// TIA Portal V20 export
// export: Created 2025-12-01T14:56:56.3805468Z, ExportSetting None, DisplayName Totally Integrated Automation Portal, DisplayVersion V20 Update 3, DisplayName TIA Portal Openness, DisplayVersion V20 Update 3, DisplayName TIA Portal Version Control Interface, DisplayVersion V20 Update 3, DisplayName STEP 7 Professional, DisplayVersion V20 Update 3, DisplayName STEP 7 Safety, DisplayVersion V20 Update 2, DisplayName WinCC Basic/Comfort/Advanced, DisplayVersion V20 Update 3, DisplayName WinCC Professional, DisplayVersion V20 Update 3, DisplayName WinCC Unified, DisplayVersion V20 Update 3
FUNCTION_BLOCK "FB490_ControlEtiquetadora_ZETES"   // FB490, LAD
{ S7_Optimized_Access := 'FALSE' }
// stored: AutoNumber false, SetENOAutomatically false
   VAR_INPUT
      NumMaquina : UInt;   // Numero de Maquina
      NumMesa : UInt;
      In_PowerOn : Bool;
      In_Online : Bool;
      In_Consumible : Bool;
      In_Bypass : Bool;
      In_BrazoRecogido : Bool;
      In_DataReady : Bool;
      In_FinCiclo : Bool;
   END_VAR
   VAR_OUTPUT
      Out_InicioCiclo : Bool;
      Parar_Tx { ExternalAccessible := 'False'; ExternalVisible := 'False'; ExternalWritable := 'False'} : Bool;
   END_VAR
   VAR
      Mx_ET00 : Bool;
      Mx_ET01 : Bool;
      Mx_ET02 : Bool;
      Mx_ET03 : Bool;
      Mx_ET04 : Bool;
      Mx_ET05 : Bool;
      Mx_ET06 : Bool;
      Mx_ET07 : Bool;
      EmpezandoProceso : Bool;
      FinalProceso : Bool;
      ErrorProceso : Bool;
      Interlock_manual { S7_SetPoint := 'True'} : "UDT_Interlock_manual_Etiquetadora";
   END_VAR
   VAR_TEMP
      VarEventos : Struct
         NumeroUT : UInt;
         ProcesoActual : UInt;
         P_EmiEventos : DWord;
         DBEventos : Word;
         NumDBEventos : UInt;
         MaxBytes : UInt;
         NumBytes : UInt;
         OffsetInicial : UInt;
         OffsetFinal : UInt;
         Conversion : DWord;
         Convertir : UInt;
         Valor : UDInt;
      END_STRUCT;
      Informe_disp_maquina : "UDT_Informe_DispositivoMaquina";
      Interlock : "UDT_Interlock_Etiquetadora_ZETES";
      retval : Int;
      cero : USInt;
      Etiq_Online : Bool;
      Etiq_Error : Bool;
      OrdenDeEtiquetar : Bool;
      Reset : Bool;
   END_VAR
   VAR_TEMP   // added for the SCL form of the ladder/FBD networks
      _w1 : Bool;
   END_VAR
BEGIN

REGION Network 1: INICIALIZAR
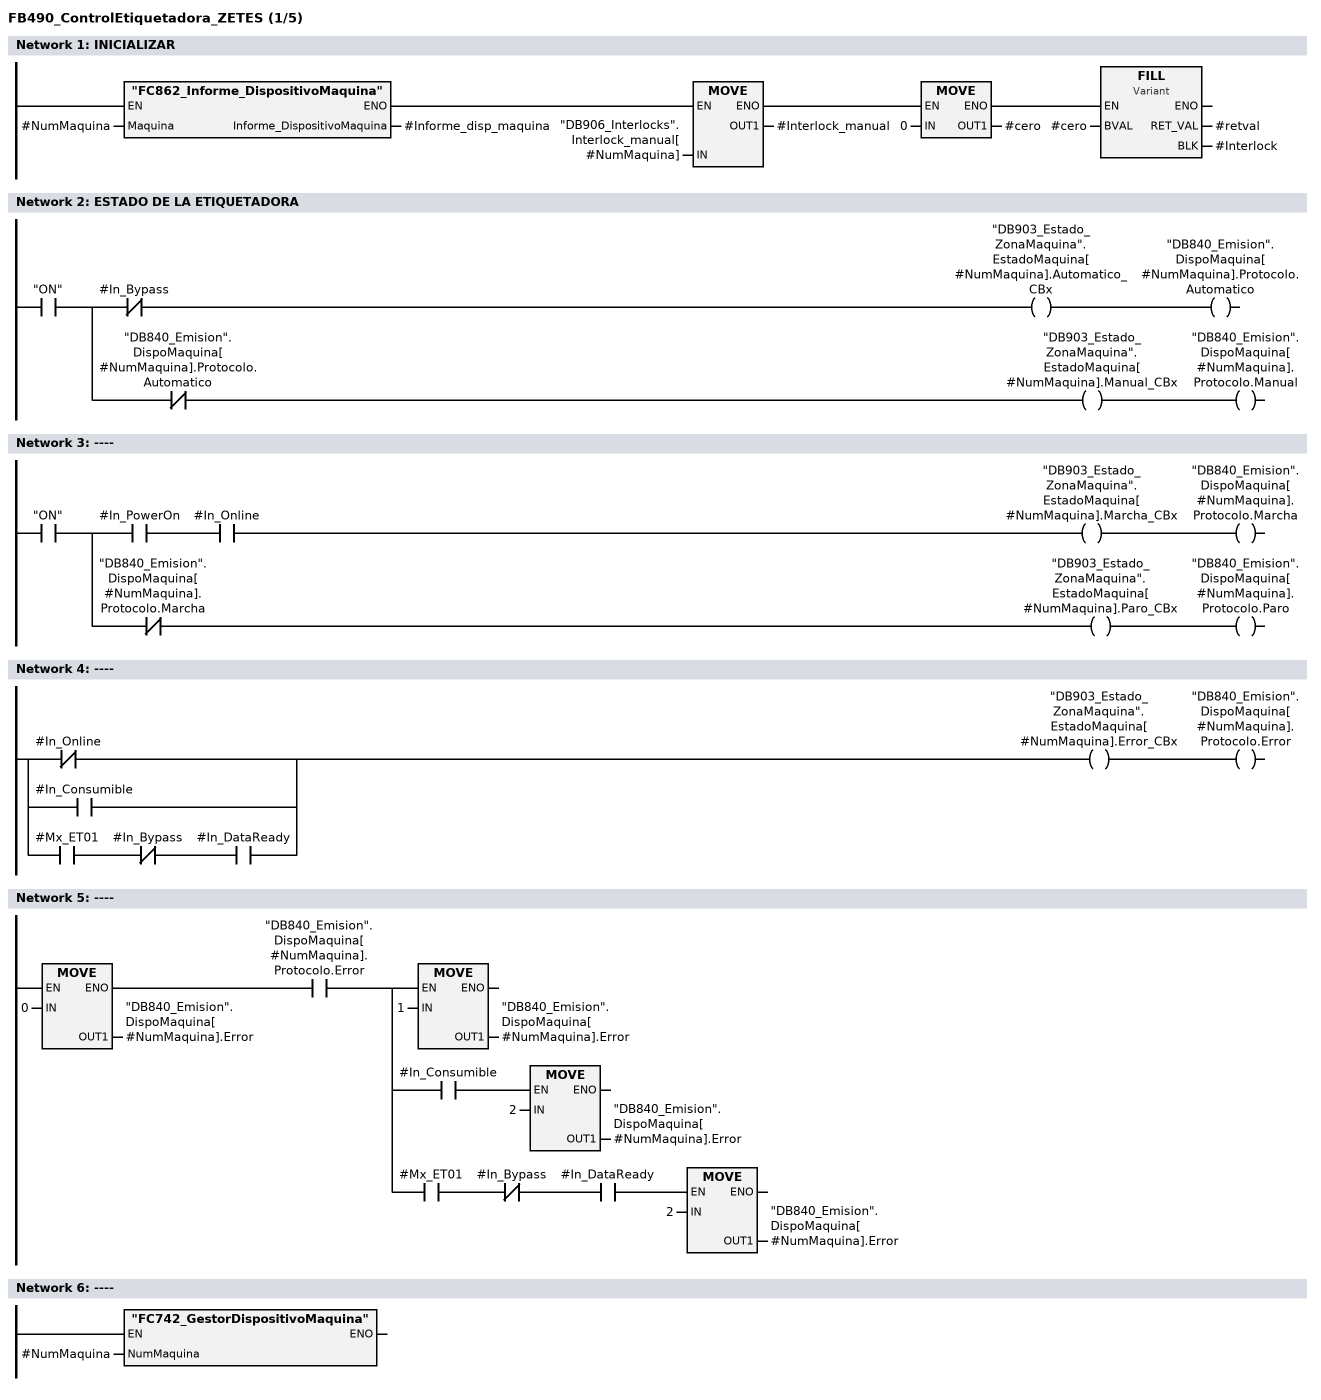
   RUNG wire#powerrail
      "FC862_Informe_DispositivoMaquina"(Maquina := #NumMaquina, Informe_DispositivoMaquina => #Informe_disp_maquina)
      Move(in := "DB906_Interlocks".Interlock_manual[#NumMaquina], out1 => #Interlock_manual)
      Move(in := 0, out1 => #cero)
      { S7_Templates := "ptr_type := Variant" } FILL(BVAL := #cero, RET_VAL => #retval, BLK => #Interlock)
   END_RUNG
   // the same network as SCL:
   "FC862_Informe_DispositivoMaquina"(Maquina := #NumMaquina,
                           Informe_DispositivoMaquina => #Informe_disp_maquina,
                           ENO => #_w1);
   IF #_w1 THEN
       #Interlock_manual := "DB906_Interlocks".Interlock_manual[#NumMaquina];
       #cero := 0;
       #retval := FILL(BVAL := #cero, BLK => #Interlock);
   END_IF;
END_REGION

REGION Network 2: ESTADO DE LA ETIQUETADORA
   RUNG wire#powerrail
      Contact( "ON" )
      wire#w1
      I_Contact( #In_Bypass )
      Coil( "DB903_Estado_ZonaMaquina".EstadoMaquina[#NumMaquina].Automatico_CBx )
      Coil( "DB840_Emision".DispoMaquina[#NumMaquina].Protocolo.Automatico )
   END_RUNG
   RUNG wire#w1
      I_Contact( "DB840_Emision".DispoMaquina[#NumMaquina].Protocolo.Automatico )
      Coil( "DB903_Estado_ZonaMaquina".EstadoMaquina[#NumMaquina].Manual_CBx )
      Coil( "DB840_Emision".DispoMaquina[#NumMaquina].Protocolo.Manual )
   END_RUNG
   // the same network as SCL:
   "DB903_Estado_ZonaMaquina".EstadoMaquina[#NumMaquina].Automatico_CBx := "ON" AND NOT #In_Bypass;
   "DB840_Emision".DispoMaquina[#NumMaquina].Protocolo.Automatico := "ON" AND NOT #In_Bypass;
   #_w1 := "ON" AND NOT "DB840_Emision".DispoMaquina[#NumMaquina].Protocolo.Automatico;
   "DB903_Estado_ZonaMaquina".EstadoMaquina[#NumMaquina].Manual_CBx := #_w1;
   "DB840_Emision".DispoMaquina[#NumMaquina].Protocolo.Manual := #_w1;
END_REGION

REGION Network 3: ----
   RUNG wire#powerrail
      Contact( "ON" )
      wire#w1
      Contact( #In_PowerOn )
      Contact( #In_Online )
      Coil( "DB903_Estado_ZonaMaquina".EstadoMaquina[#NumMaquina].Marcha_CBx )
      Coil( "DB840_Emision".DispoMaquina[#NumMaquina].Protocolo.Marcha )
   END_RUNG
   RUNG wire#w1
      I_Contact( "DB840_Emision".DispoMaquina[#NumMaquina].Protocolo.Marcha )
      Coil( "DB903_Estado_ZonaMaquina".EstadoMaquina[#NumMaquina].Paro_CBx )
      Coil( "DB840_Emision".DispoMaquina[#NumMaquina].Protocolo.Paro )
   END_RUNG
   // the same network as SCL:
   "DB903_Estado_ZonaMaquina".EstadoMaquina[#NumMaquina].Marcha_CBx := "ON" AND #In_PowerOn AND #In_Online;
   "DB840_Emision".DispoMaquina[#NumMaquina].Protocolo.Marcha := "ON" AND #In_PowerOn AND #In_Online;
   #_w1 := "ON" AND NOT "DB840_Emision".DispoMaquina[#NumMaquina].Protocolo.Marcha;
   "DB903_Estado_ZonaMaquina".EstadoMaquina[#NumMaquina].Paro_CBx := #_w1;
   "DB840_Emision".DispoMaquina[#NumMaquina].Protocolo.Paro := #_w1;
END_REGION

REGION Network 4: ----
   RUNG wire#powerrail
      I_Contact( #In_Online )
      wire#w1
      Coil( "DB903_Estado_ZonaMaquina".EstadoMaquina[#NumMaquina].Error_CBx )
      Coil( "DB840_Emision".DispoMaquina[#NumMaquina].Protocolo.Error )
   END_RUNG
   RUNG wire#powerrail
      Contact( #In_Consumible )
   END_RUNG wire#w1
   RUNG wire#powerrail
      Contact( #Mx_ET01 )
      I_Contact( #In_Bypass )
      Contact( #In_DataReady )
   END_RUNG wire#w1
   // the same network as SCL:
   "DB903_Estado_ZonaMaquina".EstadoMaquina[#NumMaquina].Error_CBx := NOT #In_Online OR #In_Consumible OR (#Mx_ET01 AND NOT #In_Bypass AND #In_DataReady);
   "DB840_Emision".DispoMaquina[#NumMaquina].Protocolo.Error := NOT #In_Online OR #In_Consumible OR (#Mx_ET01 AND NOT #In_Bypass AND #In_DataReady);
END_REGION

REGION Network 5: ----
   RUNG wire#powerrail
      Move(in := 0, out1 => "DB840_Emision".DispoMaquina[#NumMaquina].Error)
      Contact( "DB840_Emision".DispoMaquina[#NumMaquina].Protocolo.Error )
      wire#w1
      Move(in := 1, out1 => "DB840_Emision".DispoMaquina[#NumMaquina].Error)
   END_RUNG
   RUNG wire#w1
      Contact( #In_Consumible )
      Move(in := 2, out1 => "DB840_Emision".DispoMaquina[#NumMaquina].Error)
   END_RUNG
   RUNG wire#w1
      Contact( #Mx_ET01 )
      I_Contact( #In_Bypass )
      Contact( #In_DataReady )
      Move(in := 2, out1 => "DB840_Emision".DispoMaquina[#NumMaquina].Error)
   END_RUNG
   // the same network as SCL:
   "DB840_Emision".DispoMaquina[#NumMaquina].Error := 0;
   #_w1 := "DB840_Emision".DispoMaquina[#NumMaquina].Protocolo.Error;
   IF #_w1 THEN "DB840_Emision".DispoMaquina[#NumMaquina].Error := 1; END_IF;
   IF #_w1 AND #In_Consumible THEN "DB840_Emision".DispoMaquina[#NumMaquina].Error := 2; END_IF;
   IF #_w1 AND #Mx_ET01 AND NOT #In_Bypass AND #In_DataReady THEN
       "DB840_Emision".DispoMaquina[#NumMaquina].Error := 2;
   END_IF;
END_REGION

REGION Network 6: ----
   RUNG wire#powerrail
      "FC742_GestorDispositivoMaquina"(NumMaquina := #NumMaquina)
   END_RUNG
   // the same network as SCL:
   "FC742_GestorDispositivoMaquina"(NumMaquina := #NumMaquina);
END_REGION

REGION Network 7: VARIABLES INTERNAS - Etiquetadora en ONLINE / ERROR
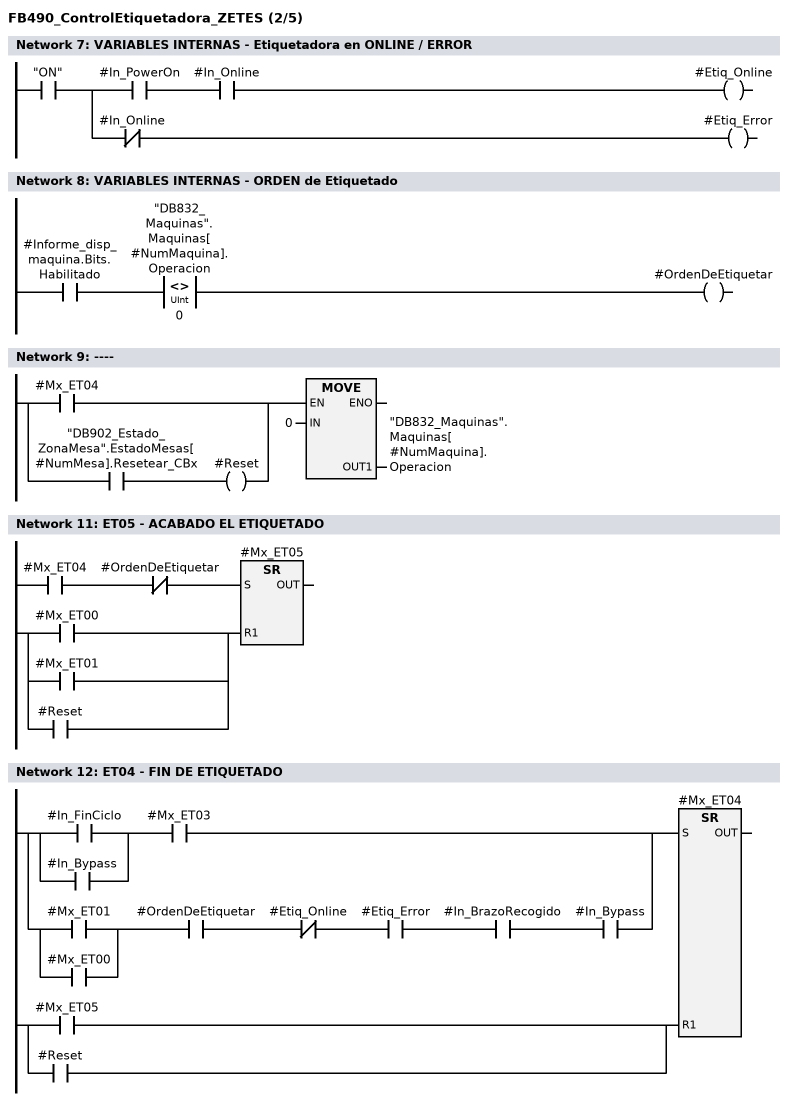
   RUNG wire#powerrail
      Contact( "ON" )
      wire#w1
      Contact( #In_PowerOn )
      Contact( #In_Online )
      Coil( #Etiq_Online )
   END_RUNG
   RUNG wire#w1
      I_Contact( #In_Online )
      Coil( #Etiq_Error )
   END_RUNG
   // the same network as SCL:
   #Etiq_Online := "ON" AND #In_PowerOn AND #In_Online;
   #Etiq_Error := "ON" AND NOT #In_Online;
END_REGION

REGION Network 8: VARIABLES INTERNAS - ORDEN de Etiquetado
   RUNG wire#powerrail
      Contact( #Informe_disp_maquina.Bits.Habilitado )
      { S7_Templates := "SrcType := UInt" } NE_Contact(in1 := "DB832_Maquinas".Maquinas[#NumMaquina].Operacion, in2 := 0)
      Coil( #OrdenDeEtiquetar )
   END_RUNG
   // the same network as SCL:
   #OrdenDeEtiquetar := #Informe_disp_maquina.Bits.Habilitado AND ("DB832_Maquinas".Maquinas[#NumMaquina].Operacion <> 0);
END_REGION

REGION Network 9: ----
   RUNG wire#powerrail
      Contact( #Mx_ET04 )
      wire#w1
      Move(in := 0, out1 => "DB832_Maquinas".Maquinas[#NumMaquina].Operacion)
   END_RUNG
   RUNG wire#powerrail
      Contact( "DB902_Estado_ZonaMesa".EstadoMesas[#NumMesa].Resetear_CBx )
      Coil( #Reset )
   END_RUNG wire#w1
   // the same network as SCL:
   #Reset := "DB902_Estado_ZonaMesa".EstadoMesas[#NumMesa].Resetear_CBx;
   IF #Mx_ET04 OR "DB902_Estado_ZonaMesa".EstadoMesas[#NumMesa].Resetear_CBx THEN
       "DB832_Maquinas".Maquinas[#NumMaquina].Operacion := 0;
   END_IF;
END_REGION

REGION Network 10: >>>>>>>>>>>>>>>>>>>>>>>>>>>>>>>>>>>>>>>>>>>>>>>>>>>>>>>>>>>>>>>>>>>>>>>>>>>>>>>>>>>>>>>>>>>>>>>
END_REGION

REGION Network 11: ET05 - ACABADO EL ETIQUETADO
   RUNG wire#powerrail
      Contact( #Mx_ET04 )
      I_Contact( #OrdenDeEtiquetar )
      S_SR(operand := #Mx_ET05, r1 := wire#w1)
   END_RUNG
   RUNG wire#powerrail
      Contact( #Mx_ET00 )
   END_RUNG wire#w1
   RUNG wire#powerrail
      Contact( #Mx_ET01 )
   END_RUNG wire#w1
   RUNG wire#powerrail
      Contact( #Reset )
   END_RUNG wire#w1
   // the same network as SCL:
   IF #Mx_ET04 AND NOT #OrdenDeEtiquetar THEN
       #Mx_ET05 := TRUE;   // SR flip-flop
   END_IF;
   IF #Mx_ET00 OR #Mx_ET01 OR #Reset THEN #Mx_ET05 := FALSE; END_IF;
END_REGION

REGION Network 12: ET04 - FIN DE ETIQUETADO
   RUNG wire#powerrail
      Contact( #In_FinCiclo )
      wire#w1
      Contact( #Mx_ET03 )
      wire#w2
      S_SR(operand := #Mx_ET04, r1 := wire#w4)
   END_RUNG
   RUNG wire#powerrail
      Contact( #In_Bypass )
   END_RUNG wire#w1
   RUNG wire#powerrail
      Contact( #Mx_ET01 )
      wire#w3
      Contact( #OrdenDeEtiquetar )
      I_Contact( #Etiq_Online )
      Contact( #Etiq_Error )
      Contact( #In_BrazoRecogido )
      Contact( #In_Bypass )
   END_RUNG wire#w2
   RUNG wire#powerrail
      Contact( #Mx_ET00 )
   END_RUNG wire#w3
   RUNG wire#powerrail
      Contact( #Mx_ET05 )
   END_RUNG wire#w4
   RUNG wire#powerrail
      Contact( #Reset )
   END_RUNG wire#w4
   // the same network as SCL:
   IF ((#In_FinCiclo OR #In_Bypass) AND #Mx_ET03) OR ((#Mx_ET01 OR #Mx_ET00) AND #OrdenDeEtiquetar AND NOT #Etiq_Online AND #Etiq_Error AND #In_BrazoRecogido AND #In_Bypass) THEN
       #Mx_ET04 := TRUE;   // SR flip-flop
   END_IF;
   IF #Mx_ET05 OR #Reset THEN #Mx_ET04 := FALSE; END_IF;
END_REGION

REGION Network 13: ET03 - ETIQUETANDO
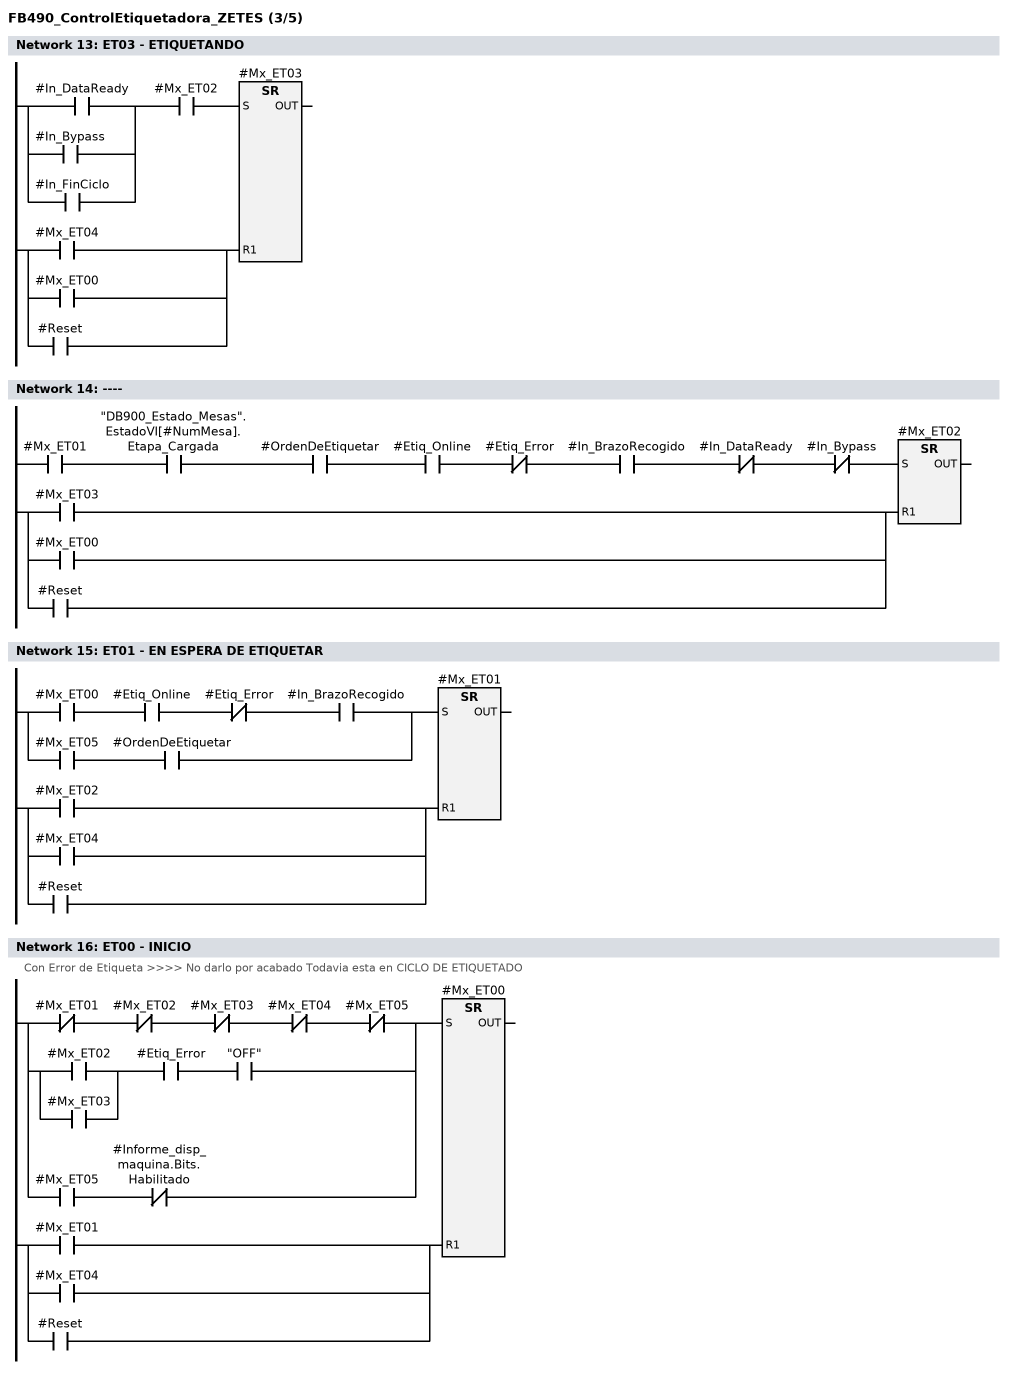
   RUNG wire#powerrail
      Contact( #In_DataReady )
      wire#w1
      Contact( #Mx_ET02 )
      S_SR(operand := #Mx_ET03, r1 := wire#w2)
   END_RUNG
   RUNG wire#powerrail
      Contact( #In_Bypass )
   END_RUNG wire#w1
   RUNG wire#powerrail
      Contact( #In_FinCiclo )
   END_RUNG wire#w1
   RUNG wire#powerrail
      Contact( #Mx_ET04 )
   END_RUNG wire#w2
   RUNG wire#powerrail
      Contact( #Mx_ET00 )
   END_RUNG wire#w2
   RUNG wire#powerrail
      Contact( #Reset )
   END_RUNG wire#w2
   // the same network as SCL:
   IF (#In_DataReady OR #In_Bypass OR #In_FinCiclo) AND #Mx_ET02 THEN
       #Mx_ET03 := TRUE;   // SR flip-flop
   END_IF;
   IF #Mx_ET04 OR #Mx_ET00 OR #Reset THEN #Mx_ET03 := FALSE; END_IF;
END_REGION

REGION Network 14: ----
   RUNG wire#powerrail
      Contact( #Mx_ET01 )
      Contact( "DB900_Estado_Mesas".EstadoVI[#NumMesa].Etapa_Cargada )
      Contact( #OrdenDeEtiquetar )
      Contact( #Etiq_Online )
      I_Contact( #Etiq_Error )
      Contact( #In_BrazoRecogido )
      I_Contact( #In_DataReady )
      I_Contact( #In_Bypass )
      S_SR(operand := #Mx_ET02, r1 := wire#w1)
   END_RUNG
   RUNG wire#powerrail
      Contact( #Mx_ET03 )
   END_RUNG wire#w1
   RUNG wire#powerrail
      Contact( #Mx_ET00 )
   END_RUNG wire#w1
   RUNG wire#powerrail
      Contact( #Reset )
   END_RUNG wire#w1
   // the same network as SCL:
   IF #Mx_ET01 AND "DB900_Estado_Mesas".EstadoVI[#NumMesa].Etapa_Cargada AND #OrdenDeEtiquetar AND #Etiq_Online AND NOT #Etiq_Error AND #In_BrazoRecogido AND NOT #In_DataReady AND NOT #In_Bypass THEN
       #Mx_ET02 := TRUE;   // SR flip-flop
   END_IF;
   IF #Mx_ET03 OR #Mx_ET00 OR #Reset THEN #Mx_ET02 := FALSE; END_IF;
END_REGION

REGION Network 15: ET01 - EN ESPERA DE ETIQUETAR
   RUNG wire#powerrail
      Contact( #Mx_ET00 )
      Contact( #Etiq_Online )
      I_Contact( #Etiq_Error )
      Contact( #In_BrazoRecogido )
      wire#w1
      S_SR(operand := #Mx_ET01, r1 := wire#w2)
   END_RUNG
   RUNG wire#powerrail
      Contact( #Mx_ET05 )
      Contact( #OrdenDeEtiquetar )
   END_RUNG wire#w1
   RUNG wire#powerrail
      Contact( #Mx_ET02 )
   END_RUNG wire#w2
   RUNG wire#powerrail
      Contact( #Mx_ET04 )
   END_RUNG wire#w2
   RUNG wire#powerrail
      Contact( #Reset )
   END_RUNG wire#w2
   // the same network as SCL:
   IF (#Mx_ET00 AND #Etiq_Online AND NOT #Etiq_Error AND #In_BrazoRecogido) OR (#Mx_ET05 AND #OrdenDeEtiquetar) THEN
       #Mx_ET01 := TRUE;   // SR flip-flop
   END_IF;
   IF #Mx_ET02 OR #Mx_ET04 OR #Reset THEN #Mx_ET01 := FALSE; END_IF;
END_REGION

REGION Network 16: ET00 - INICIO
   // Con Error de Etiqueta >>>> No darlo por acabado Todavia esta en CICLO DE ETIQUETADO
   RUNG wire#powerrail
      I_Contact( #Mx_ET01 )
      I_Contact( #Mx_ET02 )
      I_Contact( #Mx_ET03 )
      I_Contact( #Mx_ET04 )
      I_Contact( #Mx_ET05 )
      wire#w1
      S_SR(operand := #Mx_ET00, r1 := wire#w3)
   END_RUNG
   RUNG wire#powerrail
      Contact( #Mx_ET02 )
      wire#w2
      Contact( #Etiq_Error )
      Contact( "OFF" )
   END_RUNG wire#w1
   RUNG wire#powerrail
      Contact( #Mx_ET03 )
   END_RUNG wire#w2
   RUNG wire#powerrail
      Contact( #Mx_ET05 )
      I_Contact( #Informe_disp_maquina.Bits.Habilitado )
   END_RUNG wire#w1
   RUNG wire#powerrail
      Contact( #Mx_ET01 )
   END_RUNG wire#w3
   RUNG wire#powerrail
      Contact( #Mx_ET04 )
   END_RUNG wire#w3
   RUNG wire#powerrail
      Contact( #Reset )
   END_RUNG wire#w3
   // the same network as SCL:
   IF (NOT #Mx_ET01 AND NOT #Mx_ET02 AND NOT #Mx_ET03 AND NOT #Mx_ET04 AND NOT #Mx_ET05) OR ((#Mx_ET02 OR #Mx_ET03) AND #Etiq_Error AND "OFF") OR (#Mx_ET05 AND NOT #Informe_disp_maquina.Bits.Habilitado) THEN
       #Mx_ET00 := TRUE;   // SR flip-flop
   END_IF;
   IF #Mx_ET01 OR #Mx_ET04 OR #Reset THEN #Mx_ET00 := FALSE; END_IF;
END_REGION

REGION Network 17: >>>>>>>>>>>>>>>>>>>>>>>>>>>>>>>>>>>>>>>>>>>>>>>>>>>>>>>>>>>>>>>>>>>>>>>>>>>>>>>>>>>>>>>>>>>>>>>
END_REGION

REGION Network 18: VARIABLES INTERNAS - PROCESO DE ETIQUETADO >>> Eventos
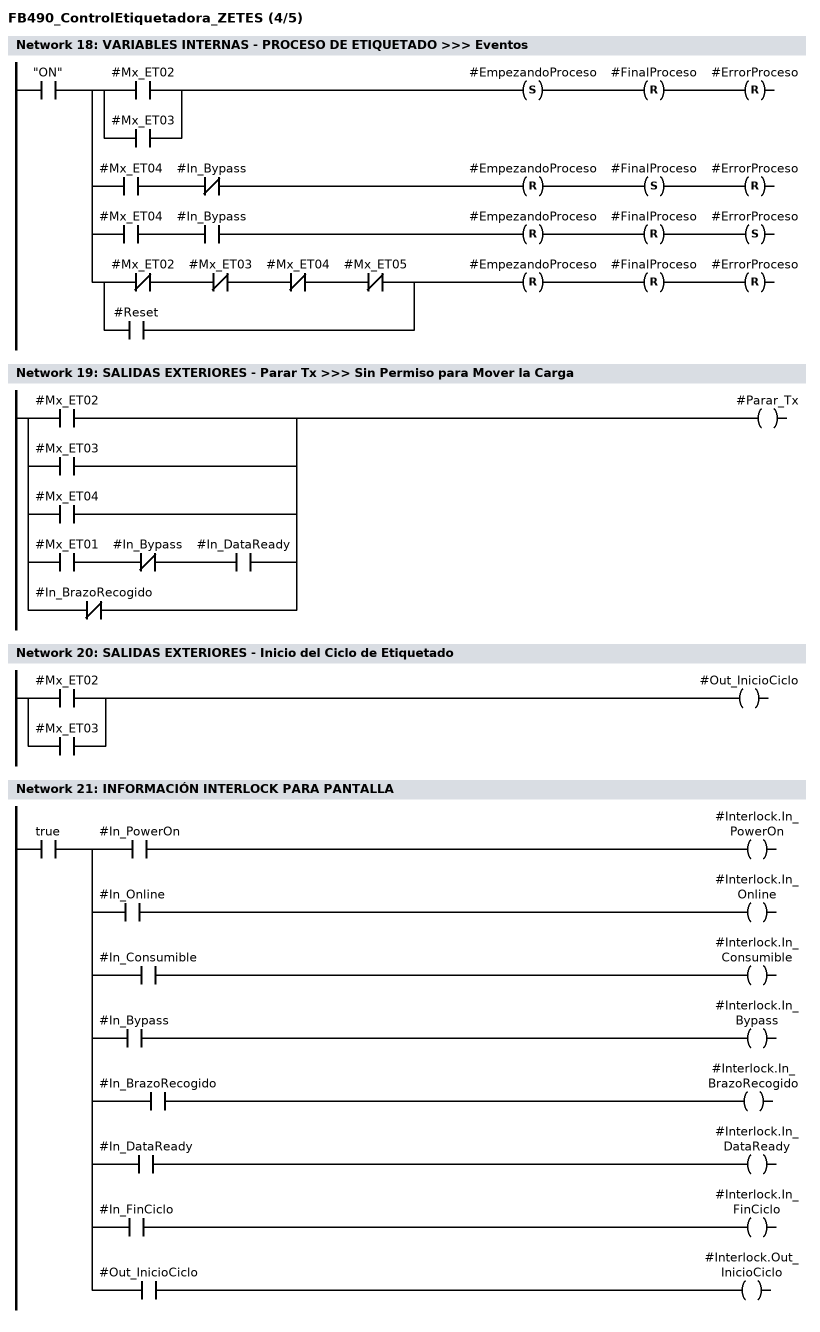
   RUNG wire#powerrail
      Contact( "ON" )
      wire#w1
      Contact( #Mx_ET02 )
      wire#w2
      S_Coil( #EmpezandoProceso )
      R_Coil( #FinalProceso )
      R_Coil( #ErrorProceso )
   END_RUNG
   RUNG wire#w1
      Contact( #Mx_ET03 )
   END_RUNG wire#w2
   RUNG wire#w1
      Contact( #Mx_ET04 )
      I_Contact( #In_Bypass )
      R_Coil( #EmpezandoProceso )
      S_Coil( #FinalProceso )
      R_Coil( #ErrorProceso )
   END_RUNG
   RUNG wire#w1
      Contact( #Mx_ET04 )
      Contact( #In_Bypass )
      R_Coil( #EmpezandoProceso )
      R_Coil( #FinalProceso )
      S_Coil( #ErrorProceso )
   END_RUNG
   RUNG wire#w1
      I_Contact( #Mx_ET02 )
      I_Contact( #Mx_ET03 )
      I_Contact( #Mx_ET04 )
      I_Contact( #Mx_ET05 )
      wire#w3
      R_Coil( #EmpezandoProceso )
      R_Coil( #FinalProceso )
      R_Coil( #ErrorProceso )
   END_RUNG
   RUNG wire#w1
      Contact( #Reset )
   END_RUNG wire#w3
   // the same network as SCL:
   IF "ON" AND (#Mx_ET02 OR #Mx_ET03) THEN
       #EmpezandoProceso := TRUE;
       #FinalProceso := FALSE;
       #ErrorProceso := FALSE;
   END_IF;
   IF "ON" AND #Mx_ET04 AND NOT #In_Bypass THEN
       #EmpezandoProceso := FALSE;
       #FinalProceso := TRUE;
       #ErrorProceso := FALSE;
   END_IF;
   IF "ON" AND #Mx_ET04 AND #In_Bypass THEN
       #EmpezandoProceso := FALSE;
       #FinalProceso := FALSE;
       #ErrorProceso := TRUE;
   END_IF;
   IF "ON" AND ((NOT #Mx_ET02 AND NOT #Mx_ET03 AND NOT #Mx_ET04 AND NOT #Mx_ET05) OR #Reset) THEN
       #EmpezandoProceso := FALSE;
       #FinalProceso := FALSE;
       #ErrorProceso := FALSE;
   END_IF;
END_REGION

REGION Network 19: SALIDAS EXTERIORES - Parar Tx >>> Sin Permiso para Mover la Carga
   RUNG wire#powerrail
      Contact( #Mx_ET02 )
      wire#w1
      Coil( #Parar_Tx )
   END_RUNG
   RUNG wire#powerrail
      Contact( #Mx_ET03 )
   END_RUNG wire#w1
   RUNG wire#powerrail
      Contact( #Mx_ET04 )
   END_RUNG wire#w1
   RUNG wire#powerrail
      Contact( #Mx_ET01 )
      I_Contact( #In_Bypass )
      Contact( #In_DataReady )
   END_RUNG wire#w1
   RUNG wire#powerrail
      I_Contact( #In_BrazoRecogido )
   END_RUNG wire#w1
   // the same network as SCL:
   #Parar_Tx := #Mx_ET02 OR #Mx_ET03 OR #Mx_ET04 OR (#Mx_ET01 AND NOT #In_Bypass AND #In_DataReady) OR NOT #In_BrazoRecogido;
END_REGION

REGION Network 20: SALIDAS EXTERIORES - Inicio del Ciclo de Etiquetado
   RUNG wire#powerrail
      Contact( #Mx_ET02 )
      wire#w1
      Coil( #Out_InicioCiclo )
   END_RUNG
   RUNG wire#powerrail
      Contact( #Mx_ET03 )
   END_RUNG wire#w1
   // the same network as SCL:
   #Out_InicioCiclo := #Mx_ET02 OR #Mx_ET03;
END_REGION

REGION Network 21: INFORMACIÓN INTERLOCK PARA PANTALLA
   RUNG wire#powerrail
      Contact( true )
      wire#w1
      Contact( #In_PowerOn )
      Coil( #Interlock.In_PowerOn )
   END_RUNG
   RUNG wire#w1
      Contact( #In_Online )
      Coil( #Interlock.In_Online )
   END_RUNG
   RUNG wire#w1
      Contact( #In_Consumible )
      Coil( #Interlock.In_Consumible )
   END_RUNG
   RUNG wire#w1
      Contact( #In_Bypass )
      Coil( #Interlock.In_Bypass )
   END_RUNG
   RUNG wire#w1
      Contact( #In_BrazoRecogido )
      Coil( #Interlock.In_BrazoRecogido )
   END_RUNG
   RUNG wire#w1
      Contact( #In_DataReady )
      Coil( #Interlock.In_DataReady )
   END_RUNG
   RUNG wire#w1
      Contact( #In_FinCiclo )
      Coil( #Interlock.In_FinCiclo )
   END_RUNG
   RUNG wire#w1
      Contact( #Out_InicioCiclo )
      Coil( #Interlock.Out_InicioCiclo )
   END_RUNG
   // the same network as SCL:
   #Interlock.In_PowerOn := true AND #In_PowerOn;
   #Interlock.In_Online := true AND #In_Online;
   #Interlock.In_Consumible := true AND #In_Consumible;
   #Interlock.In_Bypass := true AND #In_Bypass;
   #Interlock.In_BrazoRecogido := true AND #In_BrazoRecogido;
   #Interlock.In_DataReady := true AND #In_DataReady;
   #Interlock.In_FinCiclo := true AND #In_FinCiclo;
   #Interlock.Out_InicioCiclo := true AND #Out_InicioCiclo;
END_REGION

REGION Network 22: evaluar si la maquina asociada está en error para activar el error de la mesa
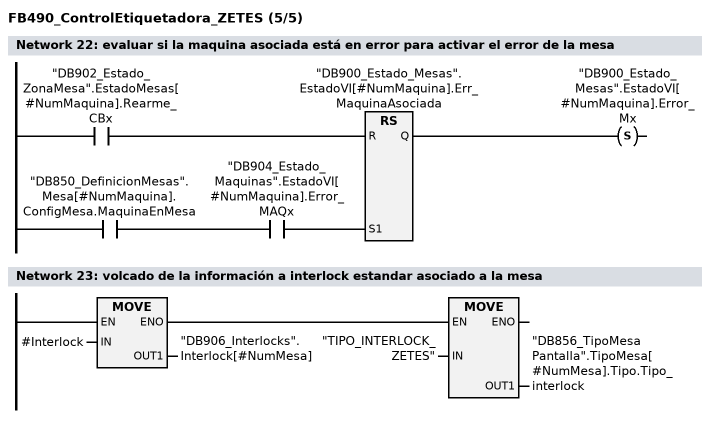
   RUNG wire#powerrail
      Contact( "DB902_Estado_ZonaMesa".EstadoMesas[#NumMaquina].Rearme_CBx )
      S_RS(operand := "DB900_Estado_Mesas".EstadoVI[#NumMaquina].Err_MaquinaAsociada, s1 := wire#w1)
      S_Coil( "DB900_Estado_Mesas".EstadoVI[#NumMaquina].Error_Mx )
   END_RUNG
   RUNG wire#powerrail
      Contact( "DB850_DefinicionMesas".Mesa[#NumMaquina].ConfigMesa.MaquinaEnMesa )
      Contact( "DB904_Estado_Maquinas".EstadoVI[#NumMaquina].Error_MAQx )
   END_RUNG wire#w1
   // the same network as SCL:
   #_w1 := "DB850_DefinicionMesas".Mesa[#NumMaquina].ConfigMesa.MaquinaEnMesa AND "DB904_Estado_Maquinas".EstadoVI[#NumMaquina].Error_MAQx;
   IF "DB902_Estado_ZonaMesa".EstadoMesas[#NumMaquina].Rearme_CBx THEN
       "DB900_Estado_Mesas".EstadoVI[#NumMaquina].Err_MaquinaAsociada := FALSE;   // RS flip-flop
   END_IF;
   IF #_w1 THEN "DB900_Estado_Mesas".EstadoVI[#NumMaquina].Err_MaquinaAsociada := TRUE; END_IF;
   IF "DB900_Estado_Mesas".EstadoVI[#NumMaquina].Err_MaquinaAsociada THEN
       "DB900_Estado_Mesas".EstadoVI[#NumMaquina].Error_Mx := TRUE;
   END_IF;
END_REGION

REGION Network 23: volcado de la información a interlock estandar asociado a la mesa
   RUNG wire#powerrail
      Move(in := #Interlock, out1 => "DB906_Interlocks".Interlock[#NumMesa])
      Move(in := "TIPO_INTERLOCK_ZETES", out1 => "DB856_TipoMesaPantalla".TipoMesa[#NumMesa].Tipo.Tipo_interlock)
   END_RUNG
   // the same network as SCL:
   "DB906_Interlocks".Interlock[#NumMesa] := #Interlock;
   "DB856_TipoMesaPantalla".TipoMesa[#NumMesa].Tipo.Tipo_interlock := "TIPO_INTERLOCK_ZETES";
END_REGION

REGION Network 24: >>>>>>>>>>>>>>>>>>>>>>>>>>>>>>>>>>>>>>>>>>>>>>>>>>>>>>>>>>>>>>>>>>>>>>>>>>>>>>>>>>>>>>>>>>>>>>>
END_REGION

NETWORK
TITLE = ENVIO DE EVENTOS - Distribucion
////////////////////////////////////////////////////////////////////////////////////
////////////////////////////////////////////////////////////////////////////////////
////////////////////////////////////////////////////////////////////////////////////
// --- Distribucion  del Estado del Proceso de la Maquina
      L     0;
      T     #VarEventos.ProcesoActual;

////////////////////////////////////////////////////////////////////////////////////
// --- Mirar que proceso es ???
      SET;
      A     #EmpezandoProceso;
      AN    #FinalProceso;
      AN    #ErrorProceso;
      JC    Es_ProcesoEmpezando;  // No Esta Empezando ?

      SET;
      AN    #EmpezandoProceso;
      A     #FinalProceso;
      AN    #ErrorProceso;
      JC    Es_ProcesoFinalizado_OK;  // No Esta Finalizado ?

      SET;
      AN    #EmpezandoProceso;
      AN    #FinalProceso;
      A     #ErrorProceso;
      JC    Es_ProcesoFinalizado_Error;  // No Esta En Error ?


// --- No Existe Proceso
      L     0;
      T     "DB832_Maquinas".Maquinas[#NumMaquina].MemoriaEstado;  // Guardo como Nuevo
      JU    Final_EmisonEvento;


////////////////////////////////////////////////////////////////////////////////////
////////////////////////////////////////////////////////////////////////////////////
////////////////////////////////////////////////////////////////////////////////////
// --- Es Inicio de Proceso
Es_ProcesoEmpezando:NOP   0;
      L     1011;  // Esta Empezando
      T     #VarEventos.ProcesoActual;
      JU    Comprobacion_EmisionEvento;


////////////////////////////////////////////////////////////////////////////////////
////////////////////////////////////////////////////////////////////////////////////
////////////////////////////////////////////////////////////////////////////////////
// --- Es Inicio de Proceso
Es_ProcesoFinalizado_OK:NOP   0;
      L     1012;  // Esta Finalizado
      T     #VarEventos.ProcesoActual;
      JU    Comprobacion_EmisionEvento;


////////////////////////////////////////////////////////////////////////////////////
////////////////////////////////////////////////////////////////////////////////////
////////////////////////////////////////////////////////////////////////////////////
// --- Es Error de Proceso
Es_ProcesoFinalizado_Error:NOP   0;
      L     1013;  // Esta En Error
      T     #VarEventos.ProcesoActual;
      JU    Comprobacion_EmisionEvento;



NETWORK
TITLE = ---- Comprobacion
////////////////////////////////////////////////////////////////////////////////////
////////////////////////////////////////////////////////////////////////////////////
////////////////////////////////////////////////////////////////////////////////////
// --- Comprobar Si hay nuevo Evento a Emitir
Comprobacion_EmisionEvento:NOP   0;
      SET;
      L     "DB832_Maquinas".Maquinas[#NumMaquina].MemoriaEstado;
      L     #VarEventos.ProcesoActual;
      ==I;
      JC    Final_EmisonEvento;  // No ha cambio de Proceso ?

      SET;
      L     0;
      L     #VarEventos.ProcesoActual;
      ==I;
      JC    Final_EmisonEvento;  // Y no sea Indetermiado ?

////////////////////////////////////////////////////////////////////////////////////
      JU    EmitirEvento;



NETWORK
TITLE = ---- Emision del Nuevo Evento
EmitirEvento:NOP   0;

////////////////////////////////////////////////////////////////////////////////////
////////////////////////////////////////////////////////////////////////////////////
////////////////////////////////////////////////////////////////////////////////////
// --- Pertenece al JDT 02 ?

      L     "JDT1_NDB_EventosEmi";
      T     #VarEventos.DBEventos;
      T     #VarEventos.NumDBEventos;
      L     "JDT1_MaxBytes";
      T     #VarEventos.MaxBytes;

      SET;
      AN    "DB850_DefinicionMesas".Mesa[#NumMesa].ConfigMesa.MesaDeJDT02;
      JC    NoJdT02;

      L     "JDT2_NDB_EventosEmi";
      T     #VarEventos.DBEventos;
      T     #VarEventos.NumDBEventos;
      L     "JDT2_MaxBytes";
      T     #VarEventos.MaxBytes;

NoJdT02:NOP   0;

////////////////////////////////////////////////////////////////////////////////////
////////////////////////////////////////////////////////////////////////////////////
////////////////////////////////////////////////////////////////////////////////////
// Inicializo el Numero de Bytes y el puntero del DB Eventos Generados
      L     0;
      T     #VarEventos.NumBytes;  // Inicializo el numero de Bytes
      LAR2;  // Inicializo el puntero de Eventos Generados

////////////////////////////////////////////////////////////////////////////////////
// Calcula el tamaño de bytes que hay en el DB Eventos Generados
      OPN   DB [#VarEventos.DBEventos];

Inicio_BusquedaFinalEventos:NOP   0;
      SET;
      L     DBB [AR2, P#0.0];
      L     0;
      ==I;
      JC    Final_BusquedaFinalEventos;  // Buscamos el final del DB = 0

      +AR2  P#1.0;
      JU    Inicio_BusquedaFinalEventos;

Final_BusquedaFinalEventos:NOP   0;
      TAR2;  // Guardo el puntero
      T     #VarEventos.P_EmiEventos;  // Sacamos el NumBytes Escritos
      SRD   3;
      T     #VarEventos.NumBytes;

////////////////////////////////////////////////////////////////////////////////////
// Comprobamos si hay sitio para mas Eventos

      L     #VarEventos.NumBytes;  // Miramos si hay sitio
      L     #VarEventos.MaxBytes;  // Max. que se pueden emitir, parametro
      >I;
      JC    Final_EmisonEvento;  // No se pueden generar más eventos



NETWORK
TITLE = ---- Formateo del Evento Del Proceso Actual
///////////////////////////////////////////////////////////////////////////////
///////////////////////////////////////////////////////////////////////////////
///////////////////////////////////////////////////////////////////////////////
// --- Formateo del Evento PROC - Estado del Proceso de la Maquina
      L     #VarEventos.P_EmiEventos;
      LAR2;  // Puntero al DB de Eventos Generados

      TAR2;  // Mirar si es el primer evento de la lista
      L     0;
      ==I;
      JC    NoEsInicio_ListaDeEventos;  // Es el primero

      OPN   DB [#VarEventos.DBEventos];
      L     ',';  // Separador entre eventos ','
      T     DBB [AR2, P#0.0];
      +AR2  P#1.0;

NoEsInicio_ListaDeEventos:NOP   0;


///////////////////////////////////////////////////////////////////////////////
///////////////////////////////////////////////////////////////////////////////
///////////////////////////////////////////////////////////////////////////////
      OPN   DB [#VarEventos.DBEventos];  // DB de Eventos Generados (A Emitir)
      L     '{';  // Inicio de Evento '{'
      T     DBB [AR2, P#0.0];
      +AR2  P#1.0;


///////////////////////////////////////////////////////////////////////////////
// --- Cuerpo del Evento PROC

      L     'DATO';  // Evento 'DATO'
      T     DBD [AR2, P#0.0];
      +AR2  P#4.0;

      L     '[';  // Evento - Atributo Proceso '[PROC]'
      T     DBB [AR2, P#0.0];
      L     'PROC';
      T     DBD [AR2, P#1.0];
      L     ']';
      T     DBB [AR2, P#5.0];
      +AR2  P#6.0;

      L     'ETIQ';  // Proceso de Etiquetado
      T     DBD [AR2, P#0.0];
      +AR2  P#4.0;


///////////////////////////////////////////////////////////////////////////////
///////////////////////////////////////////////////////////////////////////////
///////////////////////////////////////////////////////////////////////////////
      L     '[';  // Evento - Atributo MCKY '[MCKY]'
      T     DBB [AR2, P#0.0];
      L     'MCKY';
      T     DBD [AR2, P#1.0];
      L     ']';
      T     DBB [AR2, P#5.0];
      +AR2  P#6.0;

      TAR2;  // Guardar el Puntero
      T     #VarEventos.P_EmiEventos;  // Al DB de Eventos Generados

      L     "DB810_ColasMesas".Colas[#NumMesa].UT_PrimeraMesa;
      T     #VarEventos.NumeroUT;
      L     "DB812_UTs_Control".UT[#VarEventos.NumeroUT].Mckey;
      T     #VarEventos.Valor;

      L     #VarEventos.P_EmiEventos;  // Recuperar el Puntero
      LAR2;  // Al DB de Eventos Generados

// --- Convertir Valor a ASCII - Numero de Mesa
      TAR2;
      SRD   3;
      T     #VarEventos.OffsetInicial;  // Miro que offset tiene la String


      CALL  "FC893_Obtener_StringDelAtributo"
      ( DB_String := #VarEventos.NumDBEventos,
        OffsetIni := #VarEventos.OffsetInicial,
        Valor     := #VarEventos.Valor,
        OffsetFin := #VarEventos.OffsetFinal
      );  // Llamo a ObtenerStrinAtributo

      L     #VarEventos.OffsetFinal;
      SLD   3;
      LAR2;  // Recupero que offset tiene la String

///////////////////////////////////////////////////////////////////////////////
///////////////////////////////////////////////////////////////////////////////
///////////////////////////////////////////////////////////////////////////////
      OPN   DB [#VarEventos.DBEventos];  // DB de Eventos Generados (A Emitir)
      L     '[';  // Evento - Atributo MESA '[MESA]'
      T     DBB [AR2, P#0.0];
      L     'MESA';
      T     DBD [AR2, P#1.0];
      L     ']';
      T     DBB [AR2, P#5.0];
      +AR2  P#6.0;

      L     "CTE_OffsetMesa";
      L     #NumMesa;  // Numero de Maquina
      +I;
      T     #VarEventos.Valor;

// --- Convertir Valor a ASCII - Numero de Mesa
      TAR2;
      SRD   3;
      T     #VarEventos.OffsetInicial;  // Miro que offset tiene la String


      CALL  "FC893_Obtener_StringDelAtributo"
      ( DB_String := #VarEventos.NumDBEventos,
        OffsetIni := #VarEventos.OffsetInicial,
        Valor     := #VarEventos.Valor,
        OffsetFin := #VarEventos.OffsetFinal
      );  // Llamo a ObtenerStrinAtributo

      L     #VarEventos.OffsetFinal;
      SLD   3;
      LAR2;  // Recupero que offset tiene la String


///////////////////////////////////////////////////////////////////////////////
///////////////////////////////////////////////////////////////////////////////
///////////////////////////////////////////////////////////////////////////////
      OPN   DB [#VarEventos.DBEventos];  // DB de Eventos Generados (A Emitir)
      L     '[';  // Evento - Atributo Resultado '[RSLT]'
      T     DBB [AR2, P#0.0];
      L     'RSLT';
      T     DBD [AR2, P#1.0];
      L     ']';
      T     DBB [AR2, P#5.0];
      +AR2  P#6.0;

      L     #VarEventos.ProcesoActual;
      T     #VarEventos.Convertir;  // Proceso _INI o _FIN o ERRO

      CALL  "FC895_Obtener_EtiquetaDeValor"
      ( ValorEvento    := #VarEventos.Convertir,
        EtiquetaEvento := #VarEventos.Conversion
      );

      OPN   DB [#VarEventos.DBEventos];  // DB de Eventos Generados (A Emitir)
      L     #VarEventos.Conversion;
      T     DBD [AR2, P#0.0];
      +AR2  P#4.0;


///////////////////////////////////////////////////////////////////////////////
///////////////////////////////////////////////////////////////////////////////
///////////////////////////////////////////////////////////////////////////////
// --- Final del formateo del Evento

      OPN   DB [#VarEventos.DBEventos];  // DB de Eventos Generados (A Emitir)
      L     '}';  // Fin de Evento '}'
      T     DBB [AR2, P#0.0];
      +AR2  P#1.0;


///////////////////////////////////////////////////////////////////////////////
///////////////////////////////////////////////////////////////////////////////
///////////////////////////////////////////////////////////////////////////////
// --- Dar por formateado el Evento

      L     #VarEventos.ProcesoActual;  // Lo doy por tratado
      T     "DB832_Maquinas".Maquinas[#NumMaquina].MemoriaEstado;

      JU    Final_EmisonEvento;  // Ya se ha generado el evento de la Maquina

// --- Fin del Formateo del Evento de Estado del Proceso
///////////////////////////////////////////////////////////////////////////////



NETWORK
TITLE = ---- Final
///////////////////////////////////////////////////////////////////////////////
///////////////////////////////////////////////////////////////////////////////
///////////////////////////////////////////////////////////////////////////////
// --- Fin del Control
Final_EmisonEvento:NOP   0;



END_FUNCTION_BLOCK
